// TIA Portal V20 export
FUNCTION_BLOCK "Sequence_10_GaugeRnR"   // FB241, LAD
AUTHOR : ERsystem_FA2_DH. Kim
// stored: IsIECCheckEnabled true, MemoryReserve 100, Namespace Unit1.Em6, SetENOAutomatically false
   VAR_INPUT
      unitStatus { ExternalWritable := 'False'} : "LAF_typeUnitStatus";   // Unit Status used in this EM
   END_VAR
   VAR
      statSelectedJobNumber { ExternalWritable := 'False'} : DInt;   // Evaluated Job Number
      instSequenceLADStatus { ExternalWritable := 'False'} : "LAF_StatusLadSequence";
      instSequenceLADControl { ExternalWritable := 'False'} : "LAF_ControlLadSequence";
      statTonTime { ExternalAccessible := 'False'; ExternalVisible := 'False'; ExternalWritable := 'False'} : Array[0..999] of TON_TIME;
   END_VAR
   VAR CONSTANT
      STEP_IDLE : DInt := 1;
      STEP_IMMEDIATE_STOP : DInt := 9001;   // Step executed when an immediate stop command is triggered for the sequence (i.e. when unit is in state aborting)
      JOB_1_STEP_01 : DInt := 101;
      JOB_1_STEP_10 : DInt := 110;
      JOB_1_STEP_11 : DInt := 111;
      JOB_1_STEP_20 : DInt := 120;
      JOB_1_STEP_30 : DInt := 130;
      JOB_1_STEP_40 : DInt := 140;
      JOB_1_STEP_90 : DInt := 190;
      JOB_2_STEP_01 : DInt := 201;
      JOB_2_STEP_10 : DInt := 210;
      JOB_2_STEP_90 : DInt := 290;
      JOB_3_STEP_01 : DInt := 301;
      JOB_3_STEP_10 : DInt := 310;
      JOB_3_STEP_20 : DInt := 320;
      JOB_3_STEP_30 : DInt := 330;
      JOB_3_STEP_40 : DInt := 340;
      JOB_3_STEP_90 : DInt := 390;
      JOB_4_STEP_01 : DInt := 401;
      JOB_4_STEP_10 : DInt := 410;
      JOB_4_STEP_90 : DInt := 490;
   END_VAR
   VAR_TEMP   // added for the SCL form of the ladder/FBD networks
      _w1 : Bool;
   END_VAR
BEGIN

REGION Network 1: BLOCK INFO HEADER
   // (company) / (C) Copyright (year)
   // ---------------------------------------------------------------------------------
   // Title:                             (Title of this block)
   // Comment/Function: (that is implemented in the block)
   // Library/Family:           (that the source is dedicated to)
   // Author:                        (department / person in charge / contact)
   // Target System:          (test system with FW version)
   // Engineering:              TIA Portal (SW version)
   // Restrictions:               (OB types, etc.)
   // Requirements:           (hardware, technological package, etc.)
   // ---------------------------------------------------------------------------------
   // Change log table:
   // Version          | Date             | Signature      | Expert in charge  | Changes applied ------------------------|----------------------|-------------------------|--------------------------------|-----------------------
   // 001.000.000 | yyyy-mm-dd | 0x00000000 | (name of expert) | First released version
END_REGION

REGION Network 2: DESCRIPTION
   // This is a template block provided by the Automation Framework. It can be used to create an own project.
   // The Block Info Header is prepared to put in your own data.
   // Description of the block could be added here and the docu created by Code2Docu.
END_REGION

REGION Network 3: ********************* CONTROL *************************
END_REGION

REGION Network 4: Sequence Control
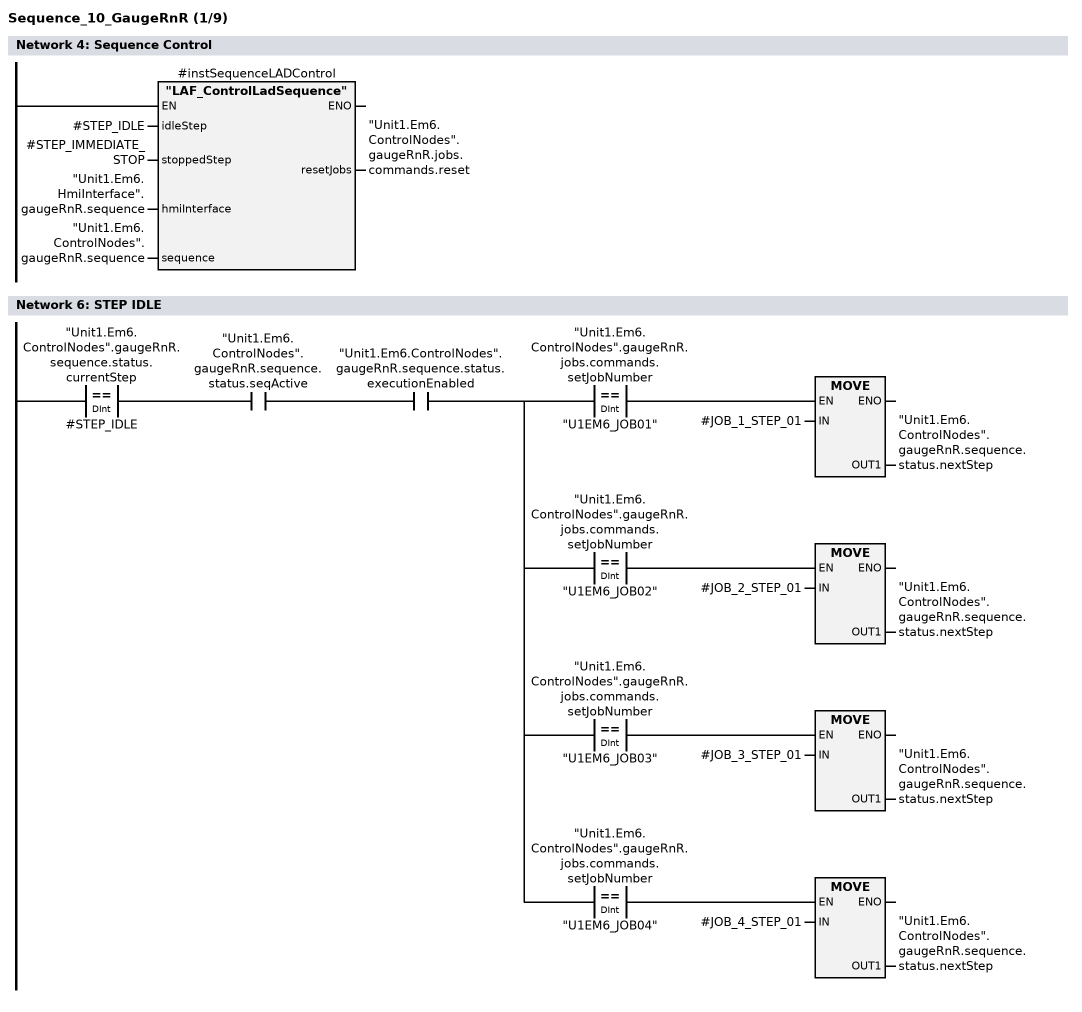
   RUNG wire#powerrail
      #instSequenceLADControl(idleStep := #STEP_IDLE, stoppedStep := #STEP_IMMEDIATE_STOP, hmiInterface := "Unit1.Em6.HmiInterface".gaugeRnR.sequence, sequence := "Unit1.Em6.ControlNodes".gaugeRnR.sequence, resetJobs => "Unit1.Em6.ControlNodes".gaugeRnR.jobs.commands.reset)
   END_RUNG
   // the same network as SCL:
   #instSequenceLADControl(idleStep := #STEP_IDLE,   // "LAF_ControlLadSequence"
                           stoppedStep := #STEP_IMMEDIATE_STOP,
                           hmiInterface := "Unit1.Em6.HmiInterface".gaugeRnR.sequence,
                           sequence := "Unit1.Em6.ControlNodes".gaugeRnR.sequence,
                           resetJobs => "Unit1.Em6.ControlNodes".gaugeRnR.jobs.commands.reset);
END_REGION

REGION Network 5: *************** JOB SELECT **************************
END_REGION

REGION Network 6: STEP IDLE
   RUNG wire#powerrail
      { S7_Templates := "SrcType := DInt" } EQ_Contact(in1 := "Unit1.Em6.ControlNodes".gaugeRnR.sequence.status.currentStep, in2 := #STEP_IDLE)
      Contact( "Unit1.Em6.ControlNodes".gaugeRnR.sequence.status.seqActive )
      Contact( "Unit1.Em6.ControlNodes".gaugeRnR.sequence.status.executionEnabled )
      wire#w1
      { S7_Templates := "SrcType := DInt" } EQ_Contact(in1 := "Unit1.Em6.ControlNodes".gaugeRnR.jobs.commands.setJobNumber, in2 := "U1EM6_JOB01")
      Move(in := #JOB_1_STEP_01, out1 => "Unit1.Em6.ControlNodes".gaugeRnR.sequence.status.nextStep)
   END_RUNG
   RUNG wire#w1
      { S7_Templates := "SrcType := DInt" } EQ_Contact(in1 := "Unit1.Em6.ControlNodes".gaugeRnR.jobs.commands.setJobNumber, in2 := "U1EM6_JOB02")
      Move(in := #JOB_2_STEP_01, out1 => "Unit1.Em6.ControlNodes".gaugeRnR.sequence.status.nextStep)
   END_RUNG
   RUNG wire#w1
      { S7_Templates := "SrcType := DInt" } EQ_Contact(in1 := "Unit1.Em6.ControlNodes".gaugeRnR.jobs.commands.setJobNumber, in2 := "U1EM6_JOB03")
      Move(in := #JOB_3_STEP_01, out1 => "Unit1.Em6.ControlNodes".gaugeRnR.sequence.status.nextStep)
   END_RUNG
   RUNG wire#w1
      { S7_Templates := "SrcType := DInt" } EQ_Contact(in1 := "Unit1.Em6.ControlNodes".gaugeRnR.jobs.commands.setJobNumber, in2 := "U1EM6_JOB04")
      Move(in := #JOB_4_STEP_01, out1 => "Unit1.Em6.ControlNodes".gaugeRnR.sequence.status.nextStep)
   END_RUNG
   // the same network as SCL:
   #_w1 := ("Unit1.Em6.ControlNodes".gaugeRnR.sequence.status.currentStep = #STEP_IDLE) AND "Unit1.Em6.ControlNodes".gaugeRnR.sequence.status.seqActive AND "Unit1.Em6.ControlNodes".gaugeRnR.sequence.status.executionEnabled;
   IF #_w1 AND ("Unit1.Em6.ControlNodes".gaugeRnR.jobs.commands.setJobNumber = "U1EM6_JOB01") THEN
       "Unit1.Em6.ControlNodes".gaugeRnR.sequence.status.nextStep := #JOB_1_STEP_01;
   END_IF;
   IF #_w1 AND ("Unit1.Em6.ControlNodes".gaugeRnR.jobs.commands.setJobNumber = "U1EM6_JOB02") THEN
       "Unit1.Em6.ControlNodes".gaugeRnR.sequence.status.nextStep := #JOB_2_STEP_01;
   END_IF;
   IF #_w1 AND ("Unit1.Em6.ControlNodes".gaugeRnR.jobs.commands.setJobNumber = "U1EM6_JOB03") THEN
       "Unit1.Em6.ControlNodes".gaugeRnR.sequence.status.nextStep := #JOB_3_STEP_01;
   END_IF;
   IF #_w1 AND ("Unit1.Em6.ControlNodes".gaugeRnR.jobs.commands.setJobNumber = "U1EM6_JOB04") THEN
       "Unit1.Em6.ControlNodes".gaugeRnR.sequence.status.nextStep := #JOB_4_STEP_01;
   END_IF;
END_REGION

REGION Network 7: *************** JOB[1] Ready ************************
END_REGION

REGION Network 8: Step[101] : JOB[1] Condition
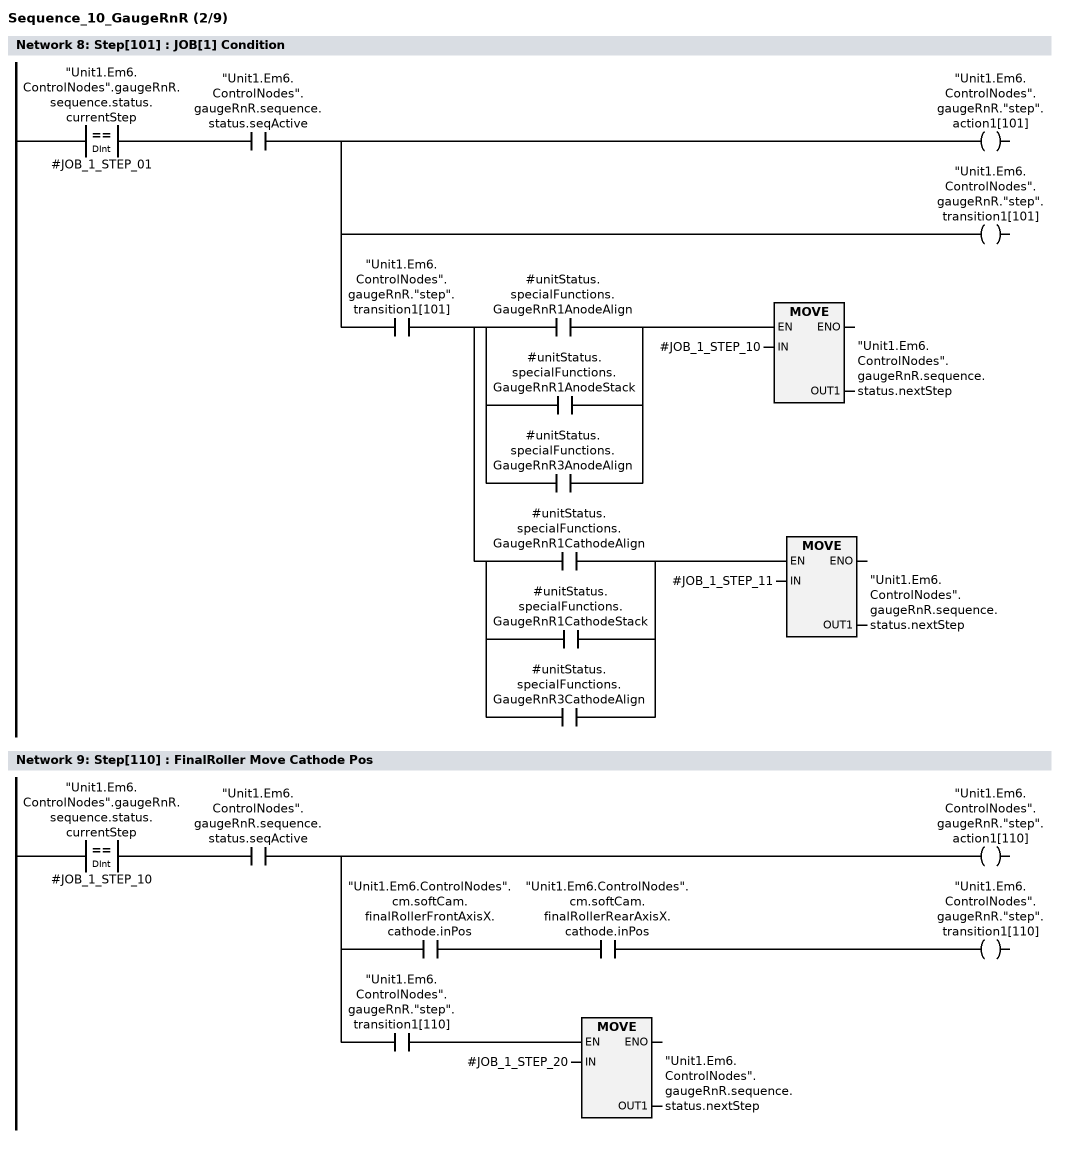
   RUNG wire#powerrail
      { S7_Templates := "SrcType := DInt" } EQ_Contact(in1 := "Unit1.Em6.ControlNodes".gaugeRnR.sequence.status.currentStep, in2 := #JOB_1_STEP_01)
      Contact( "Unit1.Em6.ControlNodes".gaugeRnR.sequence.status.seqActive )
      wire#w1
      Coil( "Unit1.Em6.ControlNodes".gaugeRnR."step".action1[101] )
   END_RUNG
   RUNG wire#w1
      Coil( "Unit1.Em6.ControlNodes".gaugeRnR."step".transition1[101] )
   END_RUNG
   RUNG wire#w1
      Contact( "Unit1.Em6.ControlNodes".gaugeRnR."step".transition1[101] )
      wire#w2
      Contact( #unitStatus.specialFunctions.GaugeRnR1AnodeAlign )
      wire#w3
      Move(in := #JOB_1_STEP_10, out1 => "Unit1.Em6.ControlNodes".gaugeRnR.sequence.status.nextStep)
   END_RUNG
   RUNG wire#w2
      Contact( #unitStatus.specialFunctions.GaugeRnR1AnodeStack )
   END_RUNG wire#w3
   RUNG wire#w2
      Contact( #unitStatus.specialFunctions.GaugeRnR3AnodeAlign )
   END_RUNG wire#w3
   RUNG wire#w2
      Contact( #unitStatus.specialFunctions.GaugeRnR1CathodeAlign )
      wire#w4
      Move(in := #JOB_1_STEP_11, out1 => "Unit1.Em6.ControlNodes".gaugeRnR.sequence.status.nextStep)
   END_RUNG
   RUNG wire#w2
      Contact( #unitStatus.specialFunctions.GaugeRnR1CathodeStack )
   END_RUNG wire#w4
   RUNG wire#w2
      Contact( #unitStatus.specialFunctions.GaugeRnR3CathodeAlign )
   END_RUNG wire#w4
   // the same network as SCL:
   "Unit1.Em6.ControlNodes".gaugeRnR."step".action1[101] := ("Unit1.Em6.ControlNodes".gaugeRnR.sequence.status.currentStep = #JOB_1_STEP_01) AND "Unit1.Em6.ControlNodes".gaugeRnR.sequence.status.seqActive;
   "Unit1.Em6.ControlNodes".gaugeRnR."step".transition1[101] := ("Unit1.Em6.ControlNodes".gaugeRnR.sequence.status.currentStep = #JOB_1_STEP_01) AND "Unit1.Em6.ControlNodes".gaugeRnR.sequence.status.seqActive;
   #_w1 := ("Unit1.Em6.ControlNodes".gaugeRnR.sequence.status.currentStep = #JOB_1_STEP_01) AND "Unit1.Em6.ControlNodes".gaugeRnR.sequence.status.seqActive AND "Unit1.Em6.ControlNodes".gaugeRnR."step".transition1[101];
   IF #_w1 AND (#unitStatus.specialFunctions.GaugeRnR1AnodeAlign OR #unitStatus.specialFunctions.GaugeRnR1AnodeStack OR #unitStatus.specialFunctions.GaugeRnR3AnodeAlign) THEN
       "Unit1.Em6.ControlNodes".gaugeRnR.sequence.status.nextStep := #JOB_1_STEP_10;
   END_IF;
   IF #_w1 AND (#unitStatus.specialFunctions.GaugeRnR1CathodeAlign OR #unitStatus.specialFunctions.GaugeRnR1CathodeStack OR #unitStatus.specialFunctions.GaugeRnR3CathodeAlign) THEN
       "Unit1.Em6.ControlNodes".gaugeRnR.sequence.status.nextStep := #JOB_1_STEP_11;
   END_IF;
END_REGION

REGION Network 9: Step[110] : FinalRoller Move Cathode Pos
   RUNG wire#powerrail
      { S7_Templates := "SrcType := DInt" } EQ_Contact(in1 := "Unit1.Em6.ControlNodes".gaugeRnR.sequence.status.currentStep, in2 := #JOB_1_STEP_10)
      Contact( "Unit1.Em6.ControlNodes".gaugeRnR.sequence.status.seqActive )
      wire#w1
      Coil( "Unit1.Em6.ControlNodes".gaugeRnR."step".action1[110] )
   END_RUNG
   RUNG wire#w1
      Contact( "Unit1.Em6.ControlNodes".cm.softCam.finalRollerFrontAxisX.cathode.inPos )
      Contact( "Unit1.Em6.ControlNodes".cm.softCam.finalRollerRearAxisX.cathode.inPos )
      Coil( "Unit1.Em6.ControlNodes".gaugeRnR."step".transition1[110] )
   END_RUNG
   RUNG wire#w1
      Contact( "Unit1.Em6.ControlNodes".gaugeRnR."step".transition1[110] )
      Move(in := #JOB_1_STEP_20, out1 => "Unit1.Em6.ControlNodes".gaugeRnR.sequence.status.nextStep)
   END_RUNG
   // the same network as SCL:
   "Unit1.Em6.ControlNodes".gaugeRnR."step".action1[110] := ("Unit1.Em6.ControlNodes".gaugeRnR.sequence.status.currentStep = #JOB_1_STEP_10) AND "Unit1.Em6.ControlNodes".gaugeRnR.sequence.status.seqActive;
   "Unit1.Em6.ControlNodes".gaugeRnR."step".transition1[110] := ("Unit1.Em6.ControlNodes".gaugeRnR.sequence.status.currentStep = #JOB_1_STEP_10) AND "Unit1.Em6.ControlNodes".gaugeRnR.sequence.status.seqActive AND "Unit1.Em6.ControlNodes".cm.softCam.finalRollerFrontAxisX.cathode.inPos AND "Unit1.Em6.ControlNodes".cm.softCam.finalRollerRearAxisX.cathode.inPos;
   IF ("Unit1.Em6.ControlNodes".gaugeRnR.sequence.status.currentStep = #JOB_1_STEP_10) AND "Unit1.Em6.ControlNodes".gaugeRnR.sequence.status.seqActive AND "Unit1.Em6.ControlNodes".gaugeRnR."step".transition1[110] THEN
       "Unit1.Em6.ControlNodes".gaugeRnR.sequence.status.nextStep := #JOB_1_STEP_20;
   END_IF;
END_REGION

REGION Network 10: Step[111] : FinalRoller Move Anode Pos
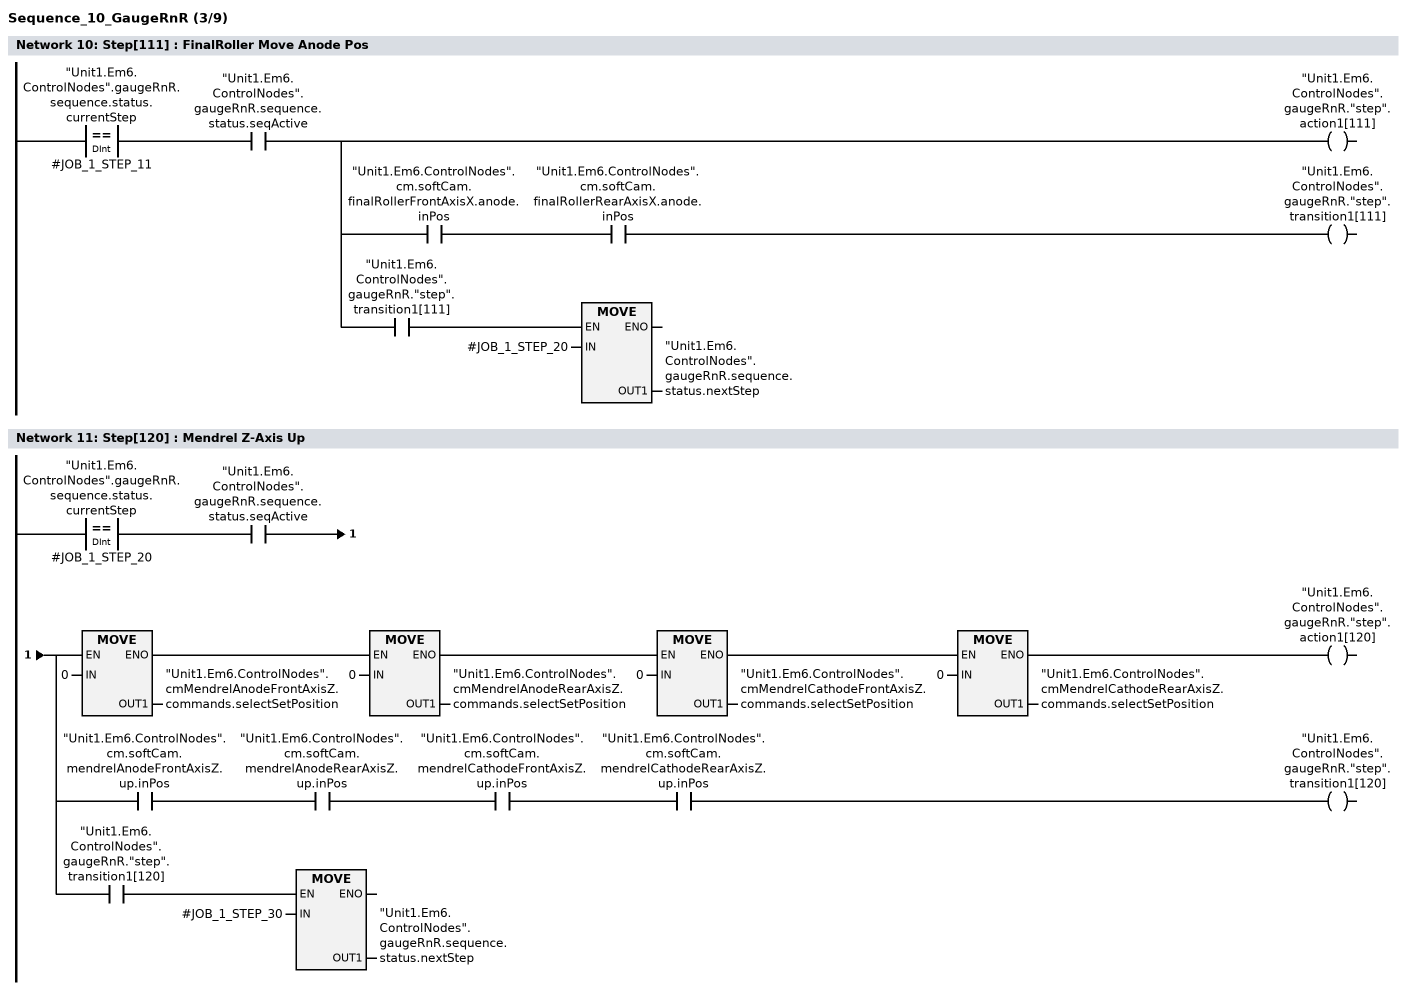
   RUNG wire#powerrail
      { S7_Templates := "SrcType := DInt" } EQ_Contact(in1 := "Unit1.Em6.ControlNodes".gaugeRnR.sequence.status.currentStep, in2 := #JOB_1_STEP_11)
      Contact( "Unit1.Em6.ControlNodes".gaugeRnR.sequence.status.seqActive )
      wire#w1
      Coil( "Unit1.Em6.ControlNodes".gaugeRnR."step".action1[111] )
   END_RUNG
   RUNG wire#w1
      Contact( "Unit1.Em6.ControlNodes".cm.softCam.finalRollerFrontAxisX.anode.inPos )
      Contact( "Unit1.Em6.ControlNodes".cm.softCam.finalRollerRearAxisX.anode.inPos )
      Coil( "Unit1.Em6.ControlNodes".gaugeRnR."step".transition1[111] )
   END_RUNG
   RUNG wire#w1
      Contact( "Unit1.Em6.ControlNodes".gaugeRnR."step".transition1[111] )
      Move(in := #JOB_1_STEP_20, out1 => "Unit1.Em6.ControlNodes".gaugeRnR.sequence.status.nextStep)
   END_RUNG
   // the same network as SCL:
   "Unit1.Em6.ControlNodes".gaugeRnR."step".action1[111] := ("Unit1.Em6.ControlNodes".gaugeRnR.sequence.status.currentStep = #JOB_1_STEP_11) AND "Unit1.Em6.ControlNodes".gaugeRnR.sequence.status.seqActive;
   "Unit1.Em6.ControlNodes".gaugeRnR."step".transition1[111] := ("Unit1.Em6.ControlNodes".gaugeRnR.sequence.status.currentStep = #JOB_1_STEP_11) AND "Unit1.Em6.ControlNodes".gaugeRnR.sequence.status.seqActive AND "Unit1.Em6.ControlNodes".cm.softCam.finalRollerFrontAxisX.anode.inPos AND "Unit1.Em6.ControlNodes".cm.softCam.finalRollerRearAxisX.anode.inPos;
   IF ("Unit1.Em6.ControlNodes".gaugeRnR.sequence.status.currentStep = #JOB_1_STEP_11) AND "Unit1.Em6.ControlNodes".gaugeRnR.sequence.status.seqActive AND "Unit1.Em6.ControlNodes".gaugeRnR."step".transition1[111] THEN
       "Unit1.Em6.ControlNodes".gaugeRnR.sequence.status.nextStep := #JOB_1_STEP_20;
   END_IF;
END_REGION

REGION Network 11: Step[120] : Mendrel Z-Axis Up
   RUNG wire#powerrail
      { S7_Templates := "SrcType := DInt" } EQ_Contact(in1 := "Unit1.Em6.ControlNodes".gaugeRnR.sequence.status.currentStep, in2 := #JOB_1_STEP_20)
      Contact( "Unit1.Em6.ControlNodes".gaugeRnR.sequence.status.seqActive )
      wire#w1
      Move(in := 0, out1 => "Unit1.Em6.ControlNodes".cmMendrelAnodeFrontAxisZ.commands.selectSetPosition)
      Move(in := 0, out1 => "Unit1.Em6.ControlNodes".cmMendrelAnodeRearAxisZ.commands.selectSetPosition)
      Move(in := 0, out1 => "Unit1.Em6.ControlNodes".cmMendrelCathodeFrontAxisZ.commands.selectSetPosition)
      Move(in := 0, out1 => "Unit1.Em6.ControlNodes".cmMendrelCathodeRearAxisZ.commands.selectSetPosition)
      Coil( "Unit1.Em6.ControlNodes".gaugeRnR."step".action1[120] )
   END_RUNG
   RUNG wire#w1
      Contact( "Unit1.Em6.ControlNodes".cm.softCam.mendrelAnodeFrontAxisZ.up.inPos )
      Contact( "Unit1.Em6.ControlNodes".cm.softCam.mendrelAnodeRearAxisZ.up.inPos )
      Contact( "Unit1.Em6.ControlNodes".cm.softCam.mendrelCathodeFrontAxisZ.up.inPos )
      Contact( "Unit1.Em6.ControlNodes".cm.softCam.mendrelCathodeRearAxisZ.up.inPos )
      Coil( "Unit1.Em6.ControlNodes".gaugeRnR."step".transition1[120] )
   END_RUNG
   RUNG wire#w1
      Contact( "Unit1.Em6.ControlNodes".gaugeRnR."step".transition1[120] )
      Move(in := #JOB_1_STEP_30, out1 => "Unit1.Em6.ControlNodes".gaugeRnR.sequence.status.nextStep)
   END_RUNG
   // the same network as SCL:
   #_w1 := ("Unit1.Em6.ControlNodes".gaugeRnR.sequence.status.currentStep = #JOB_1_STEP_20) AND "Unit1.Em6.ControlNodes".gaugeRnR.sequence.status.seqActive;
   IF #_w1 THEN
       "Unit1.Em6.ControlNodes".cmMendrelAnodeFrontAxisZ.commands.selectSetPosition := 0;
       "Unit1.Em6.ControlNodes".cmMendrelAnodeRearAxisZ.commands.selectSetPosition := 0;
       "Unit1.Em6.ControlNodes".cmMendrelCathodeFrontAxisZ.commands.selectSetPosition := 0;
       "Unit1.Em6.ControlNodes".cmMendrelCathodeRearAxisZ.commands.selectSetPosition := 0;
   END_IF;
   "Unit1.Em6.ControlNodes".gaugeRnR."step".action1[120] := #_w1;
   "Unit1.Em6.ControlNodes".gaugeRnR."step".transition1[120] := #_w1 AND "Unit1.Em6.ControlNodes".cm.softCam.mendrelAnodeFrontAxisZ.up.inPos AND "Unit1.Em6.ControlNodes".cm.softCam.mendrelAnodeRearAxisZ.up.inPos AND "Unit1.Em6.ControlNodes".cm.softCam.mendrelCathodeFrontAxisZ.up.inPos AND "Unit1.Em6.ControlNodes".cm.softCam.mendrelCathodeRearAxisZ.up.inPos;
   IF #_w1 AND "Unit1.Em6.ControlNodes".gaugeRnR."step".transition1[120] THEN
       "Unit1.Em6.ControlNodes".gaugeRnR.sequence.status.nextStep := #JOB_1_STEP_30;
   END_IF;
END_REGION

REGION Network 12: Step[130] : Mendrel Y-Axis Backward
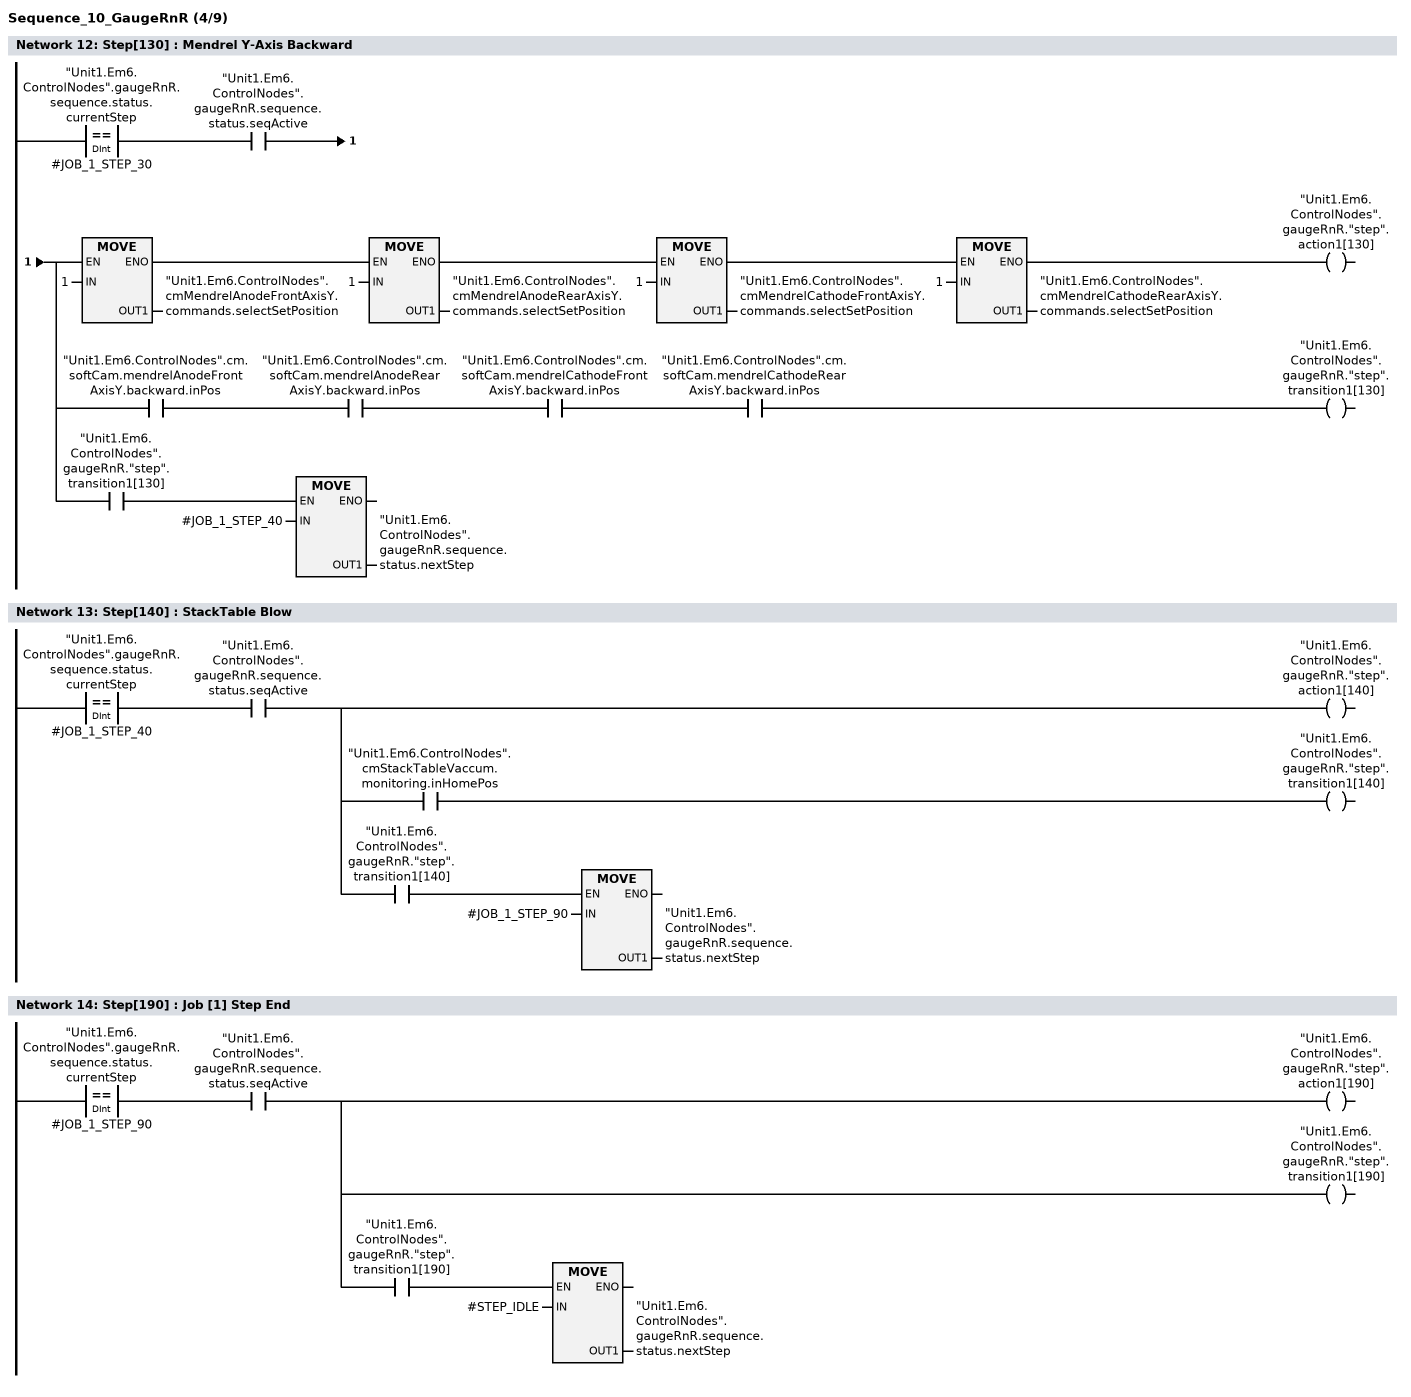
   RUNG wire#powerrail
      { S7_Templates := "SrcType := DInt" } EQ_Contact(in1 := "Unit1.Em6.ControlNodes".gaugeRnR.sequence.status.currentStep, in2 := #JOB_1_STEP_30)
      Contact( "Unit1.Em6.ControlNodes".gaugeRnR.sequence.status.seqActive )
      wire#w1
      Move(in := 1, out1 => "Unit1.Em6.ControlNodes".cmMendrelAnodeFrontAxisY.commands.selectSetPosition)
      Move(in := 1, out1 => "Unit1.Em6.ControlNodes".cmMendrelAnodeRearAxisY.commands.selectSetPosition)
      Move(in := 1, out1 => "Unit1.Em6.ControlNodes".cmMendrelCathodeFrontAxisY.commands.selectSetPosition)
      Move(in := 1, out1 => "Unit1.Em6.ControlNodes".cmMendrelCathodeRearAxisY.commands.selectSetPosition)
      Coil( "Unit1.Em6.ControlNodes".gaugeRnR."step".action1[130] )
   END_RUNG
   RUNG wire#w1
      Contact( "Unit1.Em6.ControlNodes".cm.softCam.mendrelAnodeFrontAxisY.backward.inPos )
      Contact( "Unit1.Em6.ControlNodes".cm.softCam.mendrelAnodeRearAxisY.backward.inPos )
      Contact( "Unit1.Em6.ControlNodes".cm.softCam.mendrelCathodeFrontAxisY.backward.inPos )
      Contact( "Unit1.Em6.ControlNodes".cm.softCam.mendrelCathodeRearAxisY.backward.inPos )
      Coil( "Unit1.Em6.ControlNodes".gaugeRnR."step".transition1[130] )
   END_RUNG
   RUNG wire#w1
      Contact( "Unit1.Em6.ControlNodes".gaugeRnR."step".transition1[130] )
      Move(in := #JOB_1_STEP_40, out1 => "Unit1.Em6.ControlNodes".gaugeRnR.sequence.status.nextStep)
   END_RUNG
   // the same network as SCL:
   #_w1 := ("Unit1.Em6.ControlNodes".gaugeRnR.sequence.status.currentStep = #JOB_1_STEP_30) AND "Unit1.Em6.ControlNodes".gaugeRnR.sequence.status.seqActive;
   IF #_w1 THEN
       "Unit1.Em6.ControlNodes".cmMendrelAnodeFrontAxisY.commands.selectSetPosition := 1;
       "Unit1.Em6.ControlNodes".cmMendrelAnodeRearAxisY.commands.selectSetPosition := 1;
       "Unit1.Em6.ControlNodes".cmMendrelCathodeFrontAxisY.commands.selectSetPosition := 1;
       "Unit1.Em6.ControlNodes".cmMendrelCathodeRearAxisY.commands.selectSetPosition := 1;
   END_IF;
   "Unit1.Em6.ControlNodes".gaugeRnR."step".action1[130] := #_w1;
   "Unit1.Em6.ControlNodes".gaugeRnR."step".transition1[130] := #_w1 AND "Unit1.Em6.ControlNodes".cm.softCam.mendrelAnodeFrontAxisY.backward.inPos AND "Unit1.Em6.ControlNodes".cm.softCam.mendrelAnodeRearAxisY.backward.inPos AND "Unit1.Em6.ControlNodes".cm.softCam.mendrelCathodeFrontAxisY.backward.inPos AND "Unit1.Em6.ControlNodes".cm.softCam.mendrelCathodeRearAxisY.backward.inPos;
   IF #_w1 AND "Unit1.Em6.ControlNodes".gaugeRnR."step".transition1[130] THEN
       "Unit1.Em6.ControlNodes".gaugeRnR.sequence.status.nextStep := #JOB_1_STEP_40;
   END_IF;
END_REGION

REGION Network 13: Step[140] : StackTable Blow
   RUNG wire#powerrail
      { S7_Templates := "SrcType := DInt" } EQ_Contact(in1 := "Unit1.Em6.ControlNodes".gaugeRnR.sequence.status.currentStep, in2 := #JOB_1_STEP_40)
      Contact( "Unit1.Em6.ControlNodes".gaugeRnR.sequence.status.seqActive )
      wire#w1
      Coil( "Unit1.Em6.ControlNodes".gaugeRnR."step".action1[140] )
   END_RUNG
   RUNG wire#w1
      Contact( "Unit1.Em6.ControlNodes".cmStackTableVaccum.monitoring.inHomePos )
      Coil( "Unit1.Em6.ControlNodes".gaugeRnR."step".transition1[140] )
   END_RUNG
   RUNG wire#w1
      Contact( "Unit1.Em6.ControlNodes".gaugeRnR."step".transition1[140] )
      Move(in := #JOB_1_STEP_90, out1 => "Unit1.Em6.ControlNodes".gaugeRnR.sequence.status.nextStep)
   END_RUNG
   // the same network as SCL:
   "Unit1.Em6.ControlNodes".gaugeRnR."step".action1[140] := ("Unit1.Em6.ControlNodes".gaugeRnR.sequence.status.currentStep = #JOB_1_STEP_40) AND "Unit1.Em6.ControlNodes".gaugeRnR.sequence.status.seqActive;
   "Unit1.Em6.ControlNodes".gaugeRnR."step".transition1[140] := ("Unit1.Em6.ControlNodes".gaugeRnR.sequence.status.currentStep = #JOB_1_STEP_40) AND "Unit1.Em6.ControlNodes".gaugeRnR.sequence.status.seqActive AND "Unit1.Em6.ControlNodes".cmStackTableVaccum.monitoring.inHomePos;
   IF ("Unit1.Em6.ControlNodes".gaugeRnR.sequence.status.currentStep = #JOB_1_STEP_40) AND "Unit1.Em6.ControlNodes".gaugeRnR.sequence.status.seqActive AND "Unit1.Em6.ControlNodes".gaugeRnR."step".transition1[140] THEN
       "Unit1.Em6.ControlNodes".gaugeRnR.sequence.status.nextStep := #JOB_1_STEP_90;
   END_IF;
END_REGION

REGION Network 14: Step[190] : Job [1] Step End
   RUNG wire#powerrail
      { S7_Templates := "SrcType := DInt" } EQ_Contact(in1 := "Unit1.Em6.ControlNodes".gaugeRnR.sequence.status.currentStep, in2 := #JOB_1_STEP_90)
      Contact( "Unit1.Em6.ControlNodes".gaugeRnR.sequence.status.seqActive )
      wire#w1
      Coil( "Unit1.Em6.ControlNodes".gaugeRnR."step".action1[190] )
   END_RUNG
   RUNG wire#w1
      Coil( "Unit1.Em6.ControlNodes".gaugeRnR."step".transition1[190] )
   END_RUNG
   RUNG wire#w1
      Contact( "Unit1.Em6.ControlNodes".gaugeRnR."step".transition1[190] )
      Move(in := #STEP_IDLE, out1 => "Unit1.Em6.ControlNodes".gaugeRnR.sequence.status.nextStep)
   END_RUNG
   // the same network as SCL:
   "Unit1.Em6.ControlNodes".gaugeRnR."step".action1[190] := ("Unit1.Em6.ControlNodes".gaugeRnR.sequence.status.currentStep = #JOB_1_STEP_90) AND "Unit1.Em6.ControlNodes".gaugeRnR.sequence.status.seqActive;
   "Unit1.Em6.ControlNodes".gaugeRnR."step".transition1[190] := ("Unit1.Em6.ControlNodes".gaugeRnR.sequence.status.currentStep = #JOB_1_STEP_90) AND "Unit1.Em6.ControlNodes".gaugeRnR.sequence.status.seqActive;
   IF ("Unit1.Em6.ControlNodes".gaugeRnR.sequence.status.currentStep = #JOB_1_STEP_90) AND "Unit1.Em6.ControlNodes".gaugeRnR.sequence.status.seqActive AND "Unit1.Em6.ControlNodes".gaugeRnR."step".transition1[190] THEN
       "Unit1.Em6.ControlNodes".gaugeRnR.sequence.status.nextStep := #STEP_IDLE;
   END_IF;
END_REGION

REGION Network 15: *************** JOB[2] Vaccum ************************
END_REGION

REGION Network 16: Step[201] : JOB[2] Condition
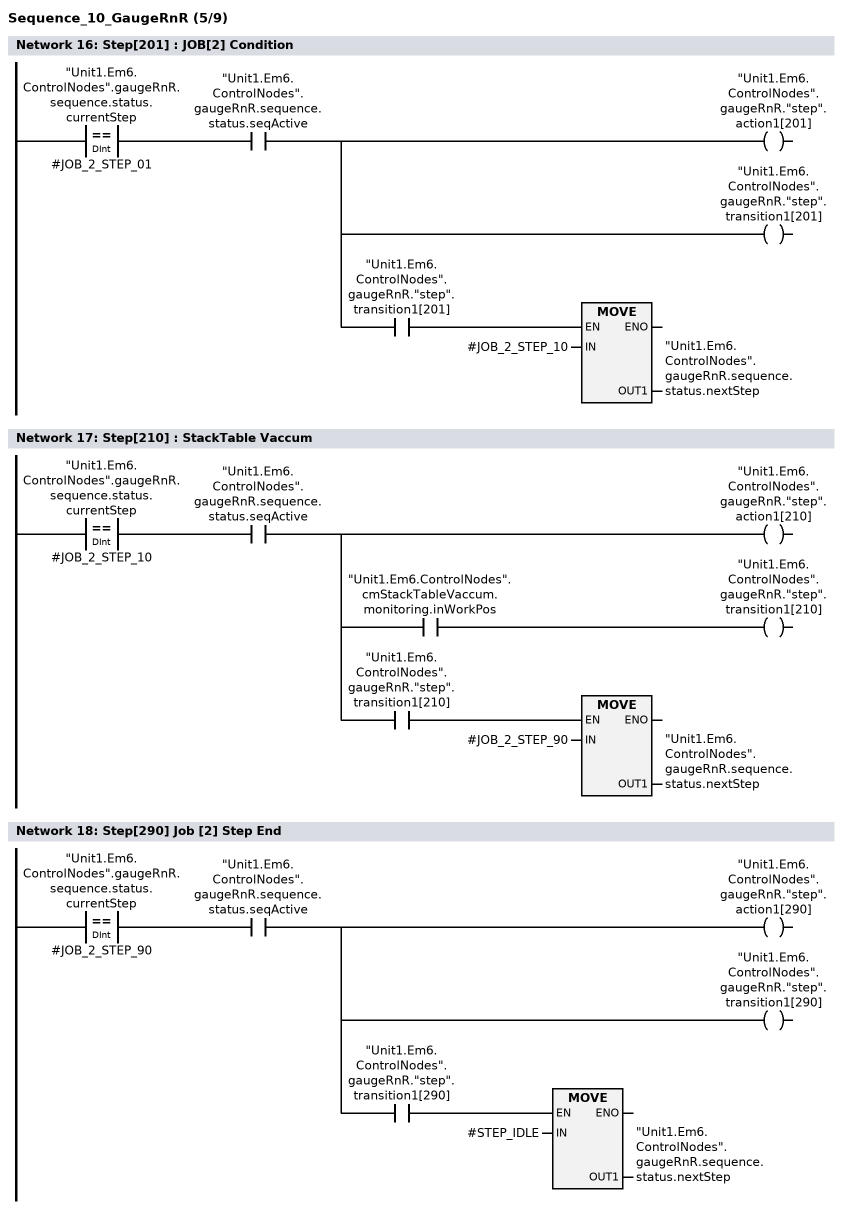
   RUNG wire#powerrail
      { S7_Templates := "SrcType := DInt" } EQ_Contact(in1 := "Unit1.Em6.ControlNodes".gaugeRnR.sequence.status.currentStep, in2 := #JOB_2_STEP_01)
      Contact( "Unit1.Em6.ControlNodes".gaugeRnR.sequence.status.seqActive )
      wire#w1
      Coil( "Unit1.Em6.ControlNodes".gaugeRnR."step".action1[201] )
   END_RUNG
   RUNG wire#w1
      Coil( "Unit1.Em6.ControlNodes".gaugeRnR."step".transition1[201] )
   END_RUNG
   RUNG wire#w1
      Contact( "Unit1.Em6.ControlNodes".gaugeRnR."step".transition1[201] )
      Move(in := #JOB_2_STEP_10, out1 => "Unit1.Em6.ControlNodes".gaugeRnR.sequence.status.nextStep)
   END_RUNG
   // the same network as SCL:
   "Unit1.Em6.ControlNodes".gaugeRnR."step".action1[201] := ("Unit1.Em6.ControlNodes".gaugeRnR.sequence.status.currentStep = #JOB_2_STEP_01) AND "Unit1.Em6.ControlNodes".gaugeRnR.sequence.status.seqActive;
   "Unit1.Em6.ControlNodes".gaugeRnR."step".transition1[201] := ("Unit1.Em6.ControlNodes".gaugeRnR.sequence.status.currentStep = #JOB_2_STEP_01) AND "Unit1.Em6.ControlNodes".gaugeRnR.sequence.status.seqActive;
   IF ("Unit1.Em6.ControlNodes".gaugeRnR.sequence.status.currentStep = #JOB_2_STEP_01) AND "Unit1.Em6.ControlNodes".gaugeRnR.sequence.status.seqActive AND "Unit1.Em6.ControlNodes".gaugeRnR."step".transition1[201] THEN
       "Unit1.Em6.ControlNodes".gaugeRnR.sequence.status.nextStep := #JOB_2_STEP_10;
   END_IF;
END_REGION

REGION Network 17: Step[210] : StackTable Vaccum
   RUNG wire#powerrail
      { S7_Templates := "SrcType := DInt" } EQ_Contact(in1 := "Unit1.Em6.ControlNodes".gaugeRnR.sequence.status.currentStep, in2 := #JOB_2_STEP_10)
      Contact( "Unit1.Em6.ControlNodes".gaugeRnR.sequence.status.seqActive )
      wire#w1
      Coil( "Unit1.Em6.ControlNodes".gaugeRnR."step".action1[210] )
   END_RUNG
   RUNG wire#w1
      Contact( "Unit1.Em6.ControlNodes".cmStackTableVaccum.monitoring.inWorkPos )
      Coil( "Unit1.Em6.ControlNodes".gaugeRnR."step".transition1[210] )
   END_RUNG
   RUNG wire#w1
      Contact( "Unit1.Em6.ControlNodes".gaugeRnR."step".transition1[210] )
      Move(in := #JOB_2_STEP_90, out1 => "Unit1.Em6.ControlNodes".gaugeRnR.sequence.status.nextStep)
   END_RUNG
   // the same network as SCL:
   "Unit1.Em6.ControlNodes".gaugeRnR."step".action1[210] := ("Unit1.Em6.ControlNodes".gaugeRnR.sequence.status.currentStep = #JOB_2_STEP_10) AND "Unit1.Em6.ControlNodes".gaugeRnR.sequence.status.seqActive;
   "Unit1.Em6.ControlNodes".gaugeRnR."step".transition1[210] := ("Unit1.Em6.ControlNodes".gaugeRnR.sequence.status.currentStep = #JOB_2_STEP_10) AND "Unit1.Em6.ControlNodes".gaugeRnR.sequence.status.seqActive AND "Unit1.Em6.ControlNodes".cmStackTableVaccum.monitoring.inWorkPos;
   IF ("Unit1.Em6.ControlNodes".gaugeRnR.sequence.status.currentStep = #JOB_2_STEP_10) AND "Unit1.Em6.ControlNodes".gaugeRnR.sequence.status.seqActive AND "Unit1.Em6.ControlNodes".gaugeRnR."step".transition1[210] THEN
       "Unit1.Em6.ControlNodes".gaugeRnR.sequence.status.nextStep := #JOB_2_STEP_90;
   END_IF;
END_REGION

REGION Network 18: Step[290] Job [2] Step End
   RUNG wire#powerrail
      { S7_Templates := "SrcType := DInt" } EQ_Contact(in1 := "Unit1.Em6.ControlNodes".gaugeRnR.sequence.status.currentStep, in2 := #JOB_2_STEP_90)
      Contact( "Unit1.Em6.ControlNodes".gaugeRnR.sequence.status.seqActive )
      wire#w1
      Coil( "Unit1.Em6.ControlNodes".gaugeRnR."step".action1[290] )
   END_RUNG
   RUNG wire#w1
      Coil( "Unit1.Em6.ControlNodes".gaugeRnR."step".transition1[290] )
   END_RUNG
   RUNG wire#w1
      Contact( "Unit1.Em6.ControlNodes".gaugeRnR."step".transition1[290] )
      Move(in := #STEP_IDLE, out1 => "Unit1.Em6.ControlNodes".gaugeRnR.sequence.status.nextStep)
   END_RUNG
   // the same network as SCL:
   "Unit1.Em6.ControlNodes".gaugeRnR."step".action1[290] := ("Unit1.Em6.ControlNodes".gaugeRnR.sequence.status.currentStep = #JOB_2_STEP_90) AND "Unit1.Em6.ControlNodes".gaugeRnR.sequence.status.seqActive;
   "Unit1.Em6.ControlNodes".gaugeRnR."step".transition1[290] := ("Unit1.Em6.ControlNodes".gaugeRnR.sequence.status.currentStep = #JOB_2_STEP_90) AND "Unit1.Em6.ControlNodes".gaugeRnR.sequence.status.seqActive;
   IF ("Unit1.Em6.ControlNodes".gaugeRnR.sequence.status.currentStep = #JOB_2_STEP_90) AND "Unit1.Em6.ControlNodes".gaugeRnR.sequence.status.seqActive AND "Unit1.Em6.ControlNodes".gaugeRnR."step".transition1[290] THEN
       "Unit1.Em6.ControlNodes".gaugeRnR.sequence.status.nextStep := #STEP_IDLE;
   END_IF;
END_REGION

REGION Network 19: *************** JOB[3] Vision ************************
END_REGION

REGION Network 20: Step[301] : JOB[3] Condition
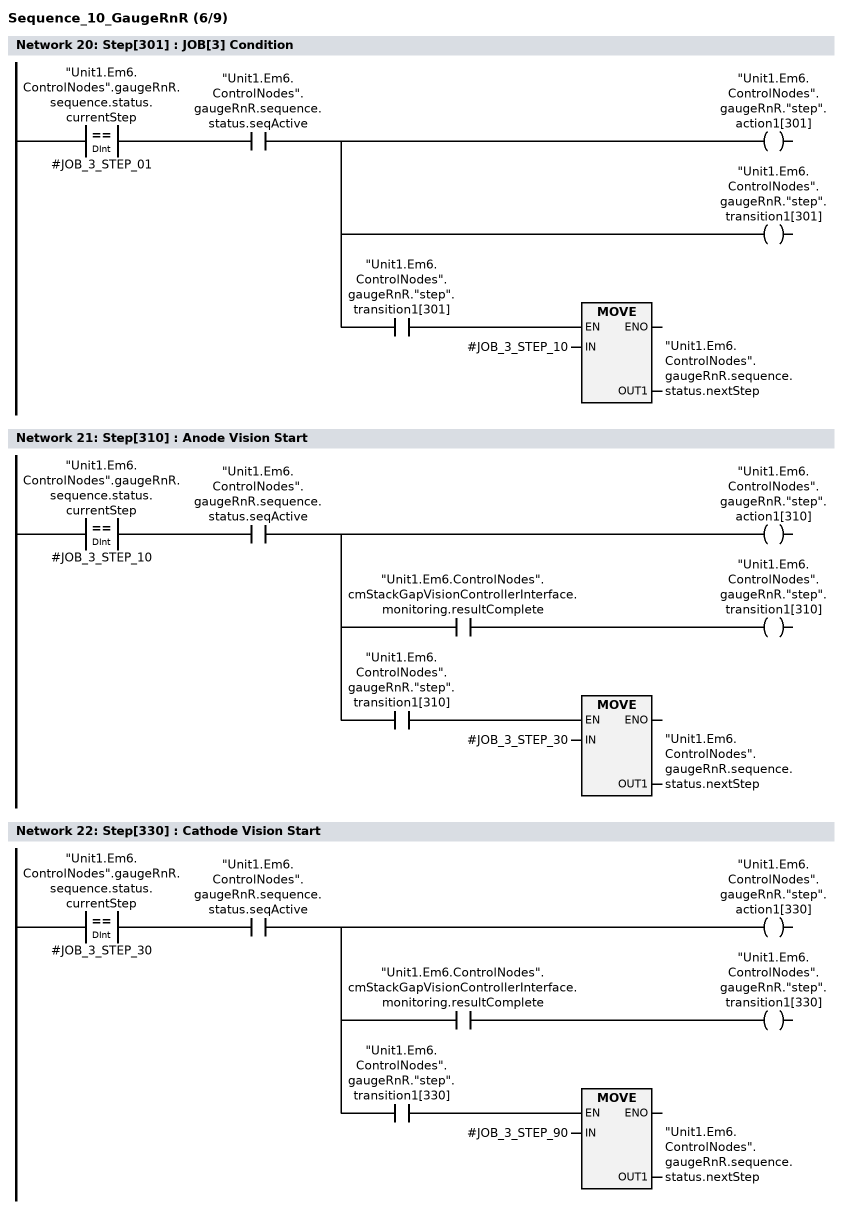
   RUNG wire#powerrail
      { S7_Templates := "SrcType := DInt" } EQ_Contact(in1 := "Unit1.Em6.ControlNodes".gaugeRnR.sequence.status.currentStep, in2 := #JOB_3_STEP_01)
      Contact( "Unit1.Em6.ControlNodes".gaugeRnR.sequence.status.seqActive )
      wire#w1
      Coil( "Unit1.Em6.ControlNodes".gaugeRnR."step".action1[301] )
   END_RUNG
   RUNG wire#w1
      Coil( "Unit1.Em6.ControlNodes".gaugeRnR."step".transition1[301] )
   END_RUNG
   RUNG wire#w1
      Contact( "Unit1.Em6.ControlNodes".gaugeRnR."step".transition1[301] )
      Move(in := #JOB_3_STEP_10, out1 => "Unit1.Em6.ControlNodes".gaugeRnR.sequence.status.nextStep)
   END_RUNG
   // the same network as SCL:
   "Unit1.Em6.ControlNodes".gaugeRnR."step".action1[301] := ("Unit1.Em6.ControlNodes".gaugeRnR.sequence.status.currentStep = #JOB_3_STEP_01) AND "Unit1.Em6.ControlNodes".gaugeRnR.sequence.status.seqActive;
   "Unit1.Em6.ControlNodes".gaugeRnR."step".transition1[301] := ("Unit1.Em6.ControlNodes".gaugeRnR.sequence.status.currentStep = #JOB_3_STEP_01) AND "Unit1.Em6.ControlNodes".gaugeRnR.sequence.status.seqActive;
   IF ("Unit1.Em6.ControlNodes".gaugeRnR.sequence.status.currentStep = #JOB_3_STEP_01) AND "Unit1.Em6.ControlNodes".gaugeRnR.sequence.status.seqActive AND "Unit1.Em6.ControlNodes".gaugeRnR."step".transition1[301] THEN
       "Unit1.Em6.ControlNodes".gaugeRnR.sequence.status.nextStep := #JOB_3_STEP_10;
   END_IF;
END_REGION

REGION Network 21: Step[310] : Anode Vision Start
   RUNG wire#powerrail
      { S7_Templates := "SrcType := DInt" } EQ_Contact(in1 := "Unit1.Em6.ControlNodes".gaugeRnR.sequence.status.currentStep, in2 := #JOB_3_STEP_10)
      Contact( "Unit1.Em6.ControlNodes".gaugeRnR.sequence.status.seqActive )
      wire#w1
      Coil( "Unit1.Em6.ControlNodes".gaugeRnR."step".action1[310] )
   END_RUNG
   RUNG wire#w1
      Contact( "Unit1.Em6.ControlNodes".cmStackGapVisionControllerInterface.monitoring.resultComplete )
      Coil( "Unit1.Em6.ControlNodes".gaugeRnR."step".transition1[310] )
   END_RUNG
   RUNG wire#w1
      Contact( "Unit1.Em6.ControlNodes".gaugeRnR."step".transition1[310] )
      Move(in := #JOB_3_STEP_30, out1 => "Unit1.Em6.ControlNodes".gaugeRnR.sequence.status.nextStep)
   END_RUNG
   // the same network as SCL:
   "Unit1.Em6.ControlNodes".gaugeRnR."step".action1[310] := ("Unit1.Em6.ControlNodes".gaugeRnR.sequence.status.currentStep = #JOB_3_STEP_10) AND "Unit1.Em6.ControlNodes".gaugeRnR.sequence.status.seqActive;
   "Unit1.Em6.ControlNodes".gaugeRnR."step".transition1[310] := ("Unit1.Em6.ControlNodes".gaugeRnR.sequence.status.currentStep = #JOB_3_STEP_10) AND "Unit1.Em6.ControlNodes".gaugeRnR.sequence.status.seqActive AND "Unit1.Em6.ControlNodes".cmStackGapVisionControllerInterface.monitoring.resultComplete;
   IF ("Unit1.Em6.ControlNodes".gaugeRnR.sequence.status.currentStep = #JOB_3_STEP_10) AND "Unit1.Em6.ControlNodes".gaugeRnR.sequence.status.seqActive AND "Unit1.Em6.ControlNodes".gaugeRnR."step".transition1[310] THEN
       "Unit1.Em6.ControlNodes".gaugeRnR.sequence.status.nextStep := #JOB_3_STEP_30;
   END_IF;
END_REGION

REGION Network 22: Step[330] : Cathode Vision Start
   RUNG wire#powerrail
      { S7_Templates := "SrcType := DInt" } EQ_Contact(in1 := "Unit1.Em6.ControlNodes".gaugeRnR.sequence.status.currentStep, in2 := #JOB_3_STEP_30)
      Contact( "Unit1.Em6.ControlNodes".gaugeRnR.sequence.status.seqActive )
      wire#w1
      Coil( "Unit1.Em6.ControlNodes".gaugeRnR."step".action1[330] )
   END_RUNG
   RUNG wire#w1
      Contact( "Unit1.Em6.ControlNodes".cmStackGapVisionControllerInterface.monitoring.resultComplete )
      Coil( "Unit1.Em6.ControlNodes".gaugeRnR."step".transition1[330] )
   END_RUNG
   RUNG wire#w1
      Contact( "Unit1.Em6.ControlNodes".gaugeRnR."step".transition1[330] )
      Move(in := #JOB_3_STEP_90, out1 => "Unit1.Em6.ControlNodes".gaugeRnR.sequence.status.nextStep)
   END_RUNG
   // the same network as SCL:
   "Unit1.Em6.ControlNodes".gaugeRnR."step".action1[330] := ("Unit1.Em6.ControlNodes".gaugeRnR.sequence.status.currentStep = #JOB_3_STEP_30) AND "Unit1.Em6.ControlNodes".gaugeRnR.sequence.status.seqActive;
   "Unit1.Em6.ControlNodes".gaugeRnR."step".transition1[330] := ("Unit1.Em6.ControlNodes".gaugeRnR.sequence.status.currentStep = #JOB_3_STEP_30) AND "Unit1.Em6.ControlNodes".gaugeRnR.sequence.status.seqActive AND "Unit1.Em6.ControlNodes".cmStackGapVisionControllerInterface.monitoring.resultComplete;
   IF ("Unit1.Em6.ControlNodes".gaugeRnR.sequence.status.currentStep = #JOB_3_STEP_30) AND "Unit1.Em6.ControlNodes".gaugeRnR.sequence.status.seqActive AND "Unit1.Em6.ControlNodes".gaugeRnR."step".transition1[330] THEN
       "Unit1.Em6.ControlNodes".gaugeRnR.sequence.status.nextStep := #JOB_3_STEP_90;
   END_IF;
END_REGION

REGION Network 23: Step[390] Job [3] Step End
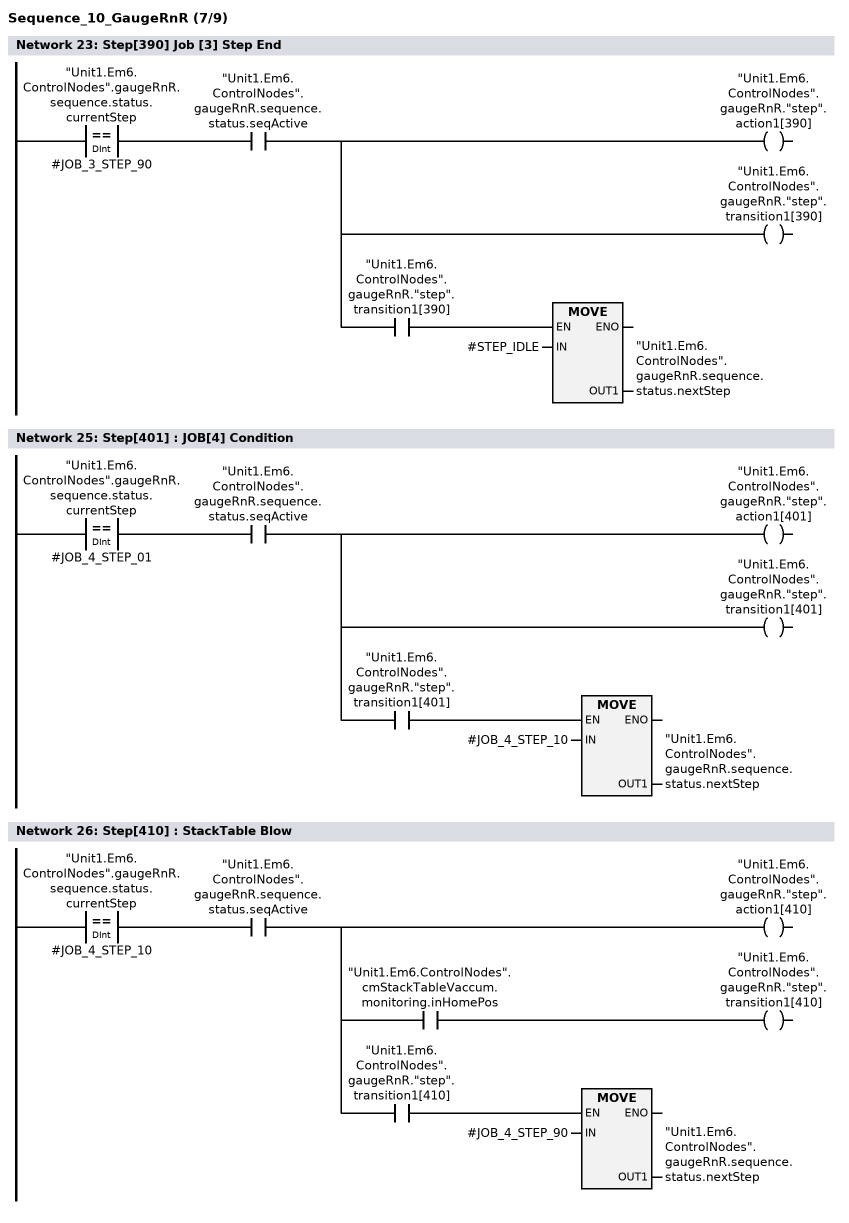
   RUNG wire#powerrail
      { S7_Templates := "SrcType := DInt" } EQ_Contact(in1 := "Unit1.Em6.ControlNodes".gaugeRnR.sequence.status.currentStep, in2 := #JOB_3_STEP_90)
      Contact( "Unit1.Em6.ControlNodes".gaugeRnR.sequence.status.seqActive )
      wire#w1
      Coil( "Unit1.Em6.ControlNodes".gaugeRnR."step".action1[390] )
   END_RUNG
   RUNG wire#w1
      Coil( "Unit1.Em6.ControlNodes".gaugeRnR."step".transition1[390] )
   END_RUNG
   RUNG wire#w1
      Contact( "Unit1.Em6.ControlNodes".gaugeRnR."step".transition1[390] )
      Move(in := #STEP_IDLE, out1 => "Unit1.Em6.ControlNodes".gaugeRnR.sequence.status.nextStep)
   END_RUNG
   // the same network as SCL:
   "Unit1.Em6.ControlNodes".gaugeRnR."step".action1[390] := ("Unit1.Em6.ControlNodes".gaugeRnR.sequence.status.currentStep = #JOB_3_STEP_90) AND "Unit1.Em6.ControlNodes".gaugeRnR.sequence.status.seqActive;
   "Unit1.Em6.ControlNodes".gaugeRnR."step".transition1[390] := ("Unit1.Em6.ControlNodes".gaugeRnR.sequence.status.currentStep = #JOB_3_STEP_90) AND "Unit1.Em6.ControlNodes".gaugeRnR.sequence.status.seqActive;
   IF ("Unit1.Em6.ControlNodes".gaugeRnR.sequence.status.currentStep = #JOB_3_STEP_90) AND "Unit1.Em6.ControlNodes".gaugeRnR.sequence.status.seqActive AND "Unit1.Em6.ControlNodes".gaugeRnR."step".transition1[390] THEN
       "Unit1.Em6.ControlNodes".gaugeRnR.sequence.status.nextStep := #STEP_IDLE;
   END_IF;
END_REGION

REGION Network 24: *************** JOB[4] Blow ************************
END_REGION

REGION Network 25: Step[401] : JOB[4] Condition
   RUNG wire#powerrail
      { S7_Templates := "SrcType := DInt" } EQ_Contact(in1 := "Unit1.Em6.ControlNodes".gaugeRnR.sequence.status.currentStep, in2 := #JOB_4_STEP_01)
      Contact( "Unit1.Em6.ControlNodes".gaugeRnR.sequence.status.seqActive )
      wire#w1
      Coil( "Unit1.Em6.ControlNodes".gaugeRnR."step".action1[401] )
   END_RUNG
   RUNG wire#w1
      Coil( "Unit1.Em6.ControlNodes".gaugeRnR."step".transition1[401] )
   END_RUNG
   RUNG wire#w1
      Contact( "Unit1.Em6.ControlNodes".gaugeRnR."step".transition1[401] )
      Move(in := #JOB_4_STEP_10, out1 => "Unit1.Em6.ControlNodes".gaugeRnR.sequence.status.nextStep)
   END_RUNG
   // the same network as SCL:
   "Unit1.Em6.ControlNodes".gaugeRnR."step".action1[401] := ("Unit1.Em6.ControlNodes".gaugeRnR.sequence.status.currentStep = #JOB_4_STEP_01) AND "Unit1.Em6.ControlNodes".gaugeRnR.sequence.status.seqActive;
   "Unit1.Em6.ControlNodes".gaugeRnR."step".transition1[401] := ("Unit1.Em6.ControlNodes".gaugeRnR.sequence.status.currentStep = #JOB_4_STEP_01) AND "Unit1.Em6.ControlNodes".gaugeRnR.sequence.status.seqActive;
   IF ("Unit1.Em6.ControlNodes".gaugeRnR.sequence.status.currentStep = #JOB_4_STEP_01) AND "Unit1.Em6.ControlNodes".gaugeRnR.sequence.status.seqActive AND "Unit1.Em6.ControlNodes".gaugeRnR."step".transition1[401] THEN
       "Unit1.Em6.ControlNodes".gaugeRnR.sequence.status.nextStep := #JOB_4_STEP_10;
   END_IF;
END_REGION

REGION Network 26: Step[410] : StackTable Blow
   RUNG wire#powerrail
      { S7_Templates := "SrcType := DInt" } EQ_Contact(in1 := "Unit1.Em6.ControlNodes".gaugeRnR.sequence.status.currentStep, in2 := #JOB_4_STEP_10)
      Contact( "Unit1.Em6.ControlNodes".gaugeRnR.sequence.status.seqActive )
      wire#w1
      Coil( "Unit1.Em6.ControlNodes".gaugeRnR."step".action1[410] )
   END_RUNG
   RUNG wire#w1
      Contact( "Unit1.Em6.ControlNodes".cmStackTableVaccum.monitoring.inHomePos )
      Coil( "Unit1.Em6.ControlNodes".gaugeRnR."step".transition1[410] )
   END_RUNG
   RUNG wire#w1
      Contact( "Unit1.Em6.ControlNodes".gaugeRnR."step".transition1[410] )
      Move(in := #JOB_4_STEP_90, out1 => "Unit1.Em6.ControlNodes".gaugeRnR.sequence.status.nextStep)
   END_RUNG
   // the same network as SCL:
   "Unit1.Em6.ControlNodes".gaugeRnR."step".action1[410] := ("Unit1.Em6.ControlNodes".gaugeRnR.sequence.status.currentStep = #JOB_4_STEP_10) AND "Unit1.Em6.ControlNodes".gaugeRnR.sequence.status.seqActive;
   "Unit1.Em6.ControlNodes".gaugeRnR."step".transition1[410] := ("Unit1.Em6.ControlNodes".gaugeRnR.sequence.status.currentStep = #JOB_4_STEP_10) AND "Unit1.Em6.ControlNodes".gaugeRnR.sequence.status.seqActive AND "Unit1.Em6.ControlNodes".cmStackTableVaccum.monitoring.inHomePos;
   IF ("Unit1.Em6.ControlNodes".gaugeRnR.sequence.status.currentStep = #JOB_4_STEP_10) AND "Unit1.Em6.ControlNodes".gaugeRnR.sequence.status.seqActive AND "Unit1.Em6.ControlNodes".gaugeRnR."step".transition1[410] THEN
       "Unit1.Em6.ControlNodes".gaugeRnR.sequence.status.nextStep := #JOB_4_STEP_90;
   END_IF;
END_REGION

REGION Network 27: Step[490] Job [4] Step End
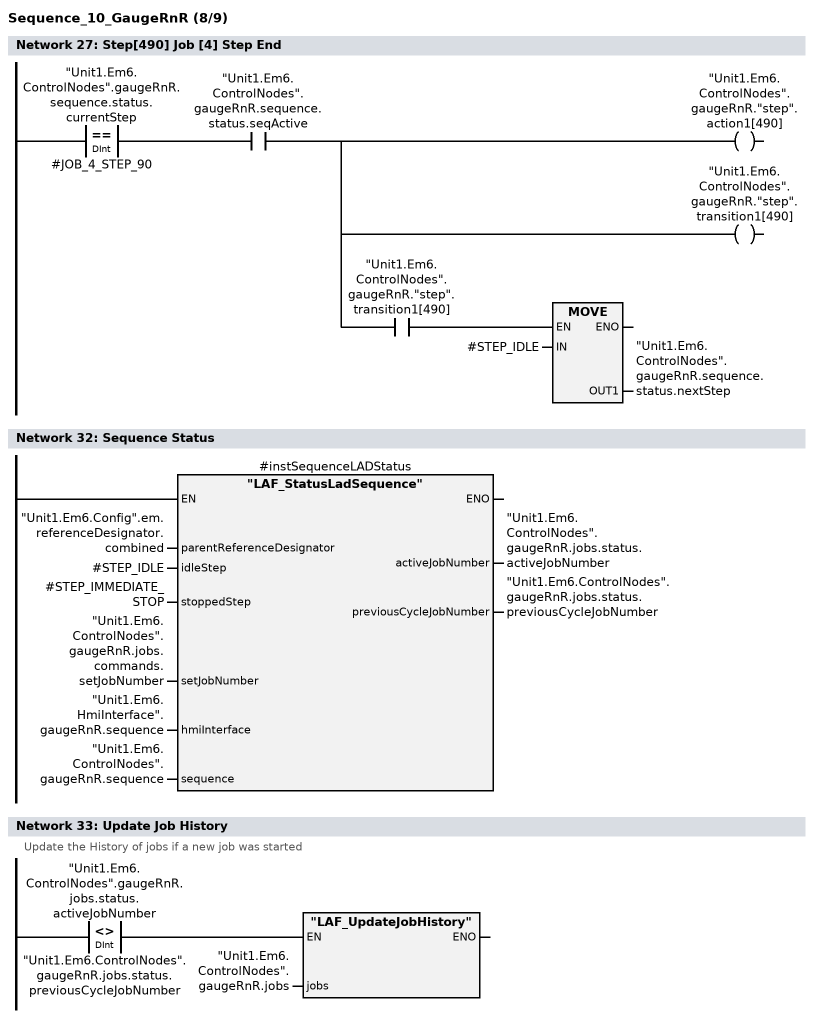
   RUNG wire#powerrail
      { S7_Templates := "SrcType := DInt" } EQ_Contact(in1 := "Unit1.Em6.ControlNodes".gaugeRnR.sequence.status.currentStep, in2 := #JOB_4_STEP_90)
      Contact( "Unit1.Em6.ControlNodes".gaugeRnR.sequence.status.seqActive )
      wire#w1
      Coil( "Unit1.Em6.ControlNodes".gaugeRnR."step".action1[490] )
   END_RUNG
   RUNG wire#w1
      Coil( "Unit1.Em6.ControlNodes".gaugeRnR."step".transition1[490] )
   END_RUNG
   RUNG wire#w1
      Contact( "Unit1.Em6.ControlNodes".gaugeRnR."step".transition1[490] )
      Move(in := #STEP_IDLE, out1 => "Unit1.Em6.ControlNodes".gaugeRnR.sequence.status.nextStep)
   END_RUNG
   // the same network as SCL:
   "Unit1.Em6.ControlNodes".gaugeRnR."step".action1[490] := ("Unit1.Em6.ControlNodes".gaugeRnR.sequence.status.currentStep = #JOB_4_STEP_90) AND "Unit1.Em6.ControlNodes".gaugeRnR.sequence.status.seqActive;
   "Unit1.Em6.ControlNodes".gaugeRnR."step".transition1[490] := ("Unit1.Em6.ControlNodes".gaugeRnR.sequence.status.currentStep = #JOB_4_STEP_90) AND "Unit1.Em6.ControlNodes".gaugeRnR.sequence.status.seqActive;
   IF ("Unit1.Em6.ControlNodes".gaugeRnR.sequence.status.currentStep = #JOB_4_STEP_90) AND "Unit1.Em6.ControlNodes".gaugeRnR.sequence.status.seqActive AND "Unit1.Em6.ControlNodes".gaugeRnR."step".transition1[490] THEN
       "Unit1.Em6.ControlNodes".gaugeRnR.sequence.status.nextStep := #STEP_IDLE;
   END_IF;
END_REGION

REGION Network 28: *************** IMMEDIATE STOP **************************
END_REGION

REGION Network 29: Immediate Stop
END_REGION

REGION Network 31: *************** Status updates **************************
END_REGION

REGION Network 32: Sequence Status
   RUNG wire#powerrail
      #instSequenceLADStatus(parentReferenceDesignator := "Unit1.Em6.Config".em.referenceDesignator.combined, idleStep := #STEP_IDLE, stoppedStep := #STEP_IMMEDIATE_STOP, setJobNumber := "Unit1.Em6.ControlNodes".gaugeRnR.jobs.commands.setJobNumber, hmiInterface := "Unit1.Em6.HmiInterface".gaugeRnR.sequence, sequence := "Unit1.Em6.ControlNodes".gaugeRnR.sequence, activeJobNumber => "Unit1.Em6.ControlNodes".gaugeRnR.jobs.status.activeJobNumber, previousCycleJobNumber => "Unit1.Em6.ControlNodes".gaugeRnR.jobs.status.previousCycleJobNumber)
   END_RUNG
   // the same network as SCL:
   #instSequenceLADStatus(parentReferenceDesignator := "Unit1.Em6.Config".em.referenceDesignator.combined,   // "LAF_StatusLadSequence"
                          idleStep := #STEP_IDLE,
                          stoppedStep := #STEP_IMMEDIATE_STOP,
                          setJobNumber := "Unit1.Em6.ControlNodes".gaugeRnR.jobs.commands.setJobNumber,
                          hmiInterface := "Unit1.Em6.HmiInterface".gaugeRnR.sequence,
                          sequence := "Unit1.Em6.ControlNodes".gaugeRnR.sequence,
                          activeJobNumber => "Unit1.Em6.ControlNodes".gaugeRnR.jobs.status.activeJobNumber,
                          previousCycleJobNumber => "Unit1.Em6.ControlNodes".gaugeRnR.jobs.status.previousCycleJobNumber);
END_REGION

REGION Network 33: Update Job History
   // Update the History of jobs if a new job was started
   RUNG wire#powerrail
      { S7_Templates := "SrcType := DInt" } NE_Contact(in1 := "Unit1.Em6.ControlNodes".gaugeRnR.jobs.status.activeJobNumber, in2 := "Unit1.Em6.ControlNodes".gaugeRnR.jobs.status.previousCycleJobNumber)
      "LAF_UpdateJobHistory"(jobs := "Unit1.Em6.ControlNodes".gaugeRnR.jobs)
   END_RUNG
   // the same network as SCL:
   IF "Unit1.Em6.ControlNodes".gaugeRnR.jobs.status.activeJobNumber <> "Unit1.Em6.ControlNodes".gaugeRnR.jobs.status.previousCycleJobNumber THEN
       "LAF_UpdateJobHistory"(jobs := "Unit1.Em6.ControlNodes".gaugeRnR.jobs);
   END_IF;
END_REGION

REGION Network 34: Output steps as String
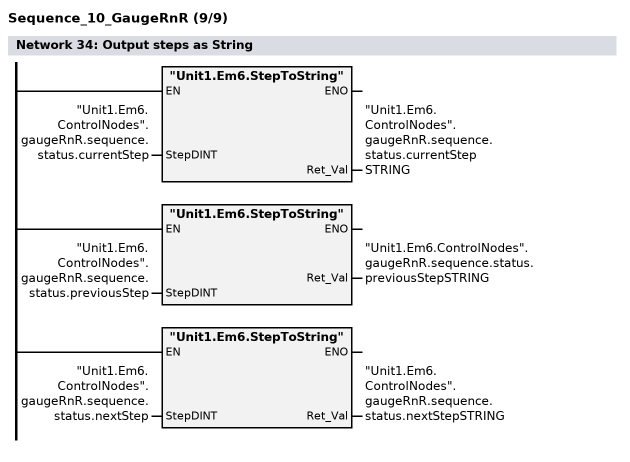
   RUNG wire#powerrail
      "Unit1.Em6.StepToString"(StepDINT := "Unit1.Em6.ControlNodes".gaugeRnR.sequence.status.currentStep, Ret_Val => "Unit1.Em6.ControlNodes".gaugeRnR.sequence.status.currentStepSTRING)
   END_RUNG
   RUNG wire#powerrail
      "Unit1.Em6.StepToString"(StepDINT := "Unit1.Em6.ControlNodes".gaugeRnR.sequence.status.previousStep, Ret_Val => "Unit1.Em6.ControlNodes".gaugeRnR.sequence.status.previousStepSTRING)
   END_RUNG
   RUNG wire#powerrail
      "Unit1.Em6.StepToString"(StepDINT := "Unit1.Em6.ControlNodes".gaugeRnR.sequence.status.nextStep, Ret_Val => "Unit1.Em6.ControlNodes".gaugeRnR.sequence.status.nextStepSTRING)
   END_RUNG
   // the same network as SCL:
   "Unit1.Em6.ControlNodes".gaugeRnR.sequence.status.currentStepSTRING := "Unit1.Em6.StepToString"(StepDINT := "Unit1.Em6.ControlNodes".gaugeRnR.sequence.status.currentStep);
   "Unit1.Em6.ControlNodes".gaugeRnR.sequence.status.previousStepSTRING := "Unit1.Em6.StepToString"(StepDINT := "Unit1.Em6.ControlNodes".gaugeRnR.sequence.status.previousStep);
   "Unit1.Em6.ControlNodes".gaugeRnR.sequence.status.nextStepSTRING := "Unit1.Em6.StepToString"(StepDINT := "Unit1.Em6.ControlNodes".gaugeRnR.sequence.status.nextStep);
END_REGION
END_FUNCTION_BLOCK
